INTERFACE ITF_HighLevelSystem

METHOD doConditionCheck : eConditionCheck
VAR_INPUT
END_VAR
END_METHOD

PROPERTY PUBLIC eCondition : eConditionCheck
GET
END_GET
SET
END_SET
END_PROPERTY

PROPERTY PUBLIC nErrorID : UDINT
GET
END_GET
SET
END_SET
END_PROPERTY

END_INTERFACE

(* stored: Version 1.1.0.1, ProductVersion 3.1.4024.12
   Itf ITF_HighLevelSystem: Id {d9a9a368-2a2c-4761-bef7-495e5c9c88bd}
   Method doConditionCheck: Id {13d88c0d-5cfb-414c-b085-09fd1b4bdec1}
   Property eCondition: Id {1f74cffe-96df-460f-bb16-9f45f604c8f8}
   Get Get: Id {55e2130a-734f-438c-a5ea-aed8c7d08a8e}
   Set Set: Id {d2c33a6c-2ee7-495e-baad-58716203d8d9}
   Property nErrorID: Id {646cf28d-12b6-4e41-aac5-c9225262184a}
   Get Get: Id {67003bea-16cc-4867-b989-2f00a77297a2}
   Set Set: Id {9f3e4eb6-a725-4d9d-a80b-c124e1388481} *)
